(* CoDeSys 2.3 library: TcSystemCX80xx.lib *)
(* Libraries: STANDARD.LIB 5.6.98 12:03:02, TcBase.lib 14.5.09 12:14:08, TcSystem.lib 27.2.12 15:08:36, TcUtilities.lib 2.3.12 19:25:40 *)

(* Global variable list: Global_Variables *)
VAR_GLOBAL
	eGlobalSUpsState	: E_S_UPS_State; (* current ups state of S-UPS *)
END_VAR

(* Data type *)
TYPE E_CX8090_LED : (
	eLED_GREEN_OFF,
	eLED_GREEN_ON,
	eLED_GREEN_FLASHING_Quick,
	eLED_GREEN_FLASHING_200ms,
	eLED_GREEN_FLASHING_500ms,
	eLED_GREEN_FLASHING_Pulse,
	eLED_RED_OFF:=20,
	eLED_RED_ON,
	eLED_RED_FLASHING_Quick,
	eLED_RED_FLASHING_200ms,
	eLED_RED_FLASHING_500ms,
	eLED_RED_FLASHING_Pulse,
	eLED_GREEN_RED_OFF:=100,
	eLED_GREEN_RED_FLASHING_200ms,
	eLED_GREEN_RED_FLASHING_500ms
);
END_TYPE

(* Data type *)
TYPE E_S_UPS_Mode : (
	eSUPS_WrPersistData_Shutdown,			(* in case of powerfailure: writing of persistent data + shutdown*)
	eSUPS_WrPersistData_NoShutdown,			(* in case of powerfailure: writing of persistent data, no shutdown*)
	eSUPS_ImmediateShutdown,				(* in case of powerfailure: skips writing of data, immediate shutdown*)
	eSUPS_CheckPowerStatus					(* in case of powerfailure: reports powerfailure without action (no writing, no shutdown) *)
);
END_TYPE

(* Data type *)
TYPE E_S_UPS_State : (
	eSUPS_StateInit := -1,
	eSUPS_PowerOK,
	eSUPS_PowerFailure,
	eSUPS_WritePersistentData,
	eSUPS_QuickShutdown,
	eSUPS_WaitForRecover,
	eSUPS_WaitForPowerOFF
);


END_TYPE

(* POU F_CX8090_LED_ERR, ST *)
FUNCTION F_CX8090_LED_ERR : INT
VAR_INPUT
	eMode	: E_CX8090_LED;
END_VAR
{library private}
VAR
	iAdr		: POINTER TO DWORD;
	UINT32Value	: DWORD;
END_VAR
F_CX8090_LED_ERR	:= eMode;

CASE eMode OF
	eLED_GREEN_OFF: 
		UINT32Value	:=0;

	eLED_GREEN_ON:
		UINT32Value	:=1;

	eLED_GREEN_FLASHING_Quick: 
		UINT32Value	:=2;

	eLED_GREEN_FLASHING_200ms: 
		UINT32Value	:=3;

	eLED_GREEN_FLASHING_500ms: 
		UINT32Value	:=16#F3;

	eLED_GREEN_FLASHING_Pulse: 
		UINT32Value	:=16#13;

	eLED_RED_OFF: 
		UINT32Value	:=0;

	eLED_RED_ON: 
		UINT32Value	:=16#1_0000;

	eLED_RED_FLASHING_Quick: 
		UINT32Value	:=16#2_0000;

	eLED_RED_FLASHING_200ms: 
		UINT32Value	:=16#3_0000;

	eLED_RED_FLASHING_500ms: 
		UINT32Value	:=16#F3_0000;

	eLED_RED_FLASHING_Pulse: 
		UINT32Value	:=16#13_0000;

	eLED_GREEN_RED_OFF:
		UINT32Value	:=0;

	eLED_GREEN_RED_FLASHING_200ms:
		UINT32Value	:=16#3_0003;

	eLED_GREEN_RED_FLASHING_500ms:
		UINT32Value	:=16#F3_00F3;
ELSE
	UINT32Value		:=0;
	F_CX8090_LED_ERR:=-1;
END_CASE

iAdr	:= 16#AA010114;
iAdr^	:= UINT32Value;
END_FUNCTION

(* POU F_CX8090_LED_WD, ST *)
FUNCTION F_CX8090_LED_WD :INT
VAR_INPUT
	eMode	: E_CX8090_LED;
END_VAR
{library private}
VAR
	iAdr  		: POINTER TO DWORD;
	UINT32Value	: DWORD;
END_VAR
F_CX8090_LED_WD := eMode;

CASE eMode OF
	eLED_GREEN_OFF: 
		UINT32Value	:=0;

	eLED_GREEN_ON:
		UINT32Value	:=1;

	eLED_GREEN_FLASHING_Quick: 
		UINT32Value	:=2;

	eLED_GREEN_FLASHING_200ms: 
		UINT32Value	:=3;

	eLED_GREEN_FLASHING_500ms: 
		UINT32Value	:=16#F3;

	eLED_GREEN_FLASHING_Pulse: 
		UINT32Value	:=16#13;

	eLED_RED_OFF: 
		UINT32Value	:=0;

	eLED_RED_ON: 
		UINT32Value	:=16#1_0000;

	eLED_RED_FLASHING_Quick: 
		UINT32Value	:=16#2_0000;

	eLED_RED_FLASHING_200ms: 
		UINT32Value	:=16#3_0000;

	eLED_RED_FLASHING_500ms: 
		UINT32Value	:=16#F3_0000;

	eLED_RED_FLASHING_Pulse: 
		UINT32Value	:=16#13_0000;

	eLED_GREEN_RED_OFF:
		UINT32Value	:=0;

	eLED_GREEN_RED_FLASHING_200ms:
		UINT32Value	:=16#3_0003;

	eLED_GREEN_RED_FLASHING_500ms:
		UINT32Value	:=16#F3_00F3;
ELSE
	UINT32Value		:=0;
	F_CX8090_LED_WD :=-1;
END_CASE

iAdr	:= 16#AA010110;
iAdr^	:= UINT32Value;
END_FUNCTION

(* POU F_CX80xx_Address, ST *)
FUNCTION F_CX80xx_Address:INT	(* Read Address switch ;Error -1 wrong CX Typ*)
VAR_INPUT
	iCX_Typ	: INT;		(*Typ of CX8000, only the number, CX8031 Typ = 8031 ...*)
END_VAR
{library private}
VAR
	iAdr  			: POINTER TO DWORD;
	UINT64Value		: DWORD;
	UINT64Value_1	: DWORD;
	UINT64Value_2	: DWORD;
	byAddress		: BYTE;
	i				: SINT;
	M_1				: BOOL;
END_VAR
iAdr		:= 16#AA000310;
UINT64Value := iAdr^;

CASE iCX_Typ OF
	8031, 8051:
		UINT64Value_1	:= 16#F-(16#F AND ROR(UINT64Value,16));
		UINT64Value_2	:= 16#F-(16#F AND ROR(UINT64Value,20));
		F_CX80xx_Address:= DWORD_TO_INT((UINT64Value_1*10+UINT64Value_2));

	8010, 8090, 8091, 8093, 8095:
		UINT64Value_2	:=16#3FF-(16#3FF AND ROR(UINT64Value,16));
		UINT64Value_1	:=0;
		FOR i:=0 TO 9 DO
			M_1 := GETBIT32(UINT64Value_2,i);
			IF M_1 THEN
				UINT64Value_1 := SETBIT32(UINT64Value_1,9-i);
			END_IF
		END_FOR
		F_CX80xx_Address := DWORD_TO_INT(UINT64Value_1);
ELSE
	F_CX80xx_Address := -1;
END_CASE
END_FUNCTION

(* POU F_GetVersionTcSystemCX80xx, ST *)
FUNCTION F_GetVersionTcSystemCX80xx : UINT
VAR_INPUT
	nVersionElement		:	INT;
END_VAR
(*
	Possible nVersionElement parameter:
	1	:	major number
	2	:	minor number
	3	:	revision number
*)
VAR
END_VAR
(* Version history:
Date        | Version    | created under      		| Author   		| Remark 
--------------------------------------------------------------------------------------------------------------------------------------------------------------------- 
2011/12/06  | 1.0.0      | V2.11.0 (Build 2040)		| ICh		    | first version
2012/04/13  | 1.0.1      | V2.11.0 (Build 2218)		| RV	      	| add LED
2012/04/17  | 1.0.2      | V2.11.0 (Build 2219)		| ICH	      	| adding Pulse to LED enum, cleanup
*) 
CASE nVersionElement OF
1:	(* major number *)
	F_GetVersionTcSystemCX80xx := 1;
2:	(* minor number *)
	F_GetVersionTcSystemCX80xx := 0;
3:	(* revision number *)
	F_GetVersionTcSystemCX80xx := 2;
ELSE
	F_GetVersionTcSystemCX80xx := 16#FFFF;
END_CASE
END_FUNCTION

(* POU FB_NT_QuickShutdown, ST *)
FUNCTION_BLOCK FB_NT_QuickShutdown
VAR_INPUT
	NETID				:T_AmsNetId;
	START				:BOOL;
	TMOUT				:TIME := DEFAULT_ADS_TIMEOUT;
END_VAR
VAR_OUTPUT
	BUSY				:BOOL;
	ERR					:BOOL;
	ERRID				:UDINT;
END_VAR
{library private}
VAR
	ADSWRTCTL1			:ADSWRTCTL;
	RisingEdge			:R_TRIG;
	DELAY				:DWORD := 16#FFFFFFFF;
END_VAR
RisingEdge(CLK:=START);

IF RisingEdge.Q THEN
	ADSWRTCTL1(	NETID := NETID,
					PORT := AMSPORT_R3_SYSSERV,
					ADSSTATE := ADSSTATE_POWERFAILURE,
					DEVSTATE := 0,
					LEN := SIZEOF(DELAY),
					SRCADDR :=ADR(DELAY),
					Write := TRUE,
					TMOUT := TMOUT
				);
ELSE
	ADSWRTCTL1( Write:=FALSE);
END_IF


BUSY := ADSWRTCTL1.BUSY;
ERR := ADSWRTCTL1.ERR;
ERRID := ADSWRTCTL1.ERRID;
END_FUNCTION_BLOCK

(* POU FB_S_UPS_CX80xx, ST *)
FUNCTION_BLOCK FB_S_UPS_CX80xx
VAR_INPUT
	sNetID					: T_AmsNetId 		:= ''; 								(* '' = local netid *)
	iPLCPort				: UINT 				:= AMSPORT_R0_PLC_RTS1;				(* PLC Runtime System for writing persistent data *)
	tTimeout				: TIME 				:= DEFAULT_ADS_TIMEOUT;				(* ADS Timeout *)
	eUpsMode				: E_S_UPS_Mode		:= eSUPS_WrPersistData_Shutdown;	(* UPS mode (w/wo writing persistent data, w/wo shutdown) *)
	ePersistentMode			: E_PersistentMode	:= SPDM_2PASS;						(* mode for writing persistent data *)
	tRecoverTime			: TIME 				:= T#10s;							(* ON time to recover from short power failure in mode eSUPS_WrPersistData_NoShutdown/eSUPS_CheckPowerStatus  *)
END_VAR
VAR_OUTPUT
	bPowerFailDetect		: BOOL;													(* TRUE while powerfailure is detected *)
	eState					: E_S_UPS_State		:= eSUPS_PowerOK;					(* current ups state *)
END_VAR
{library private}
VAR
	fbWritePersistentData	: FB_WritePersistentData;
	fbNT_QuickShutdown 		: FB_NT_QuickShutdown;
	dwTemp					: DWORD;
	WaitForOffTimer			: TON;
	bFirstCycle				: BOOL := TRUE;
	bPowerOKInFirstCycle	: BOOL := FALSE;
	iAdr 					: POINTER TO DWORD := 16#B78A4000;
END_VAR
(* monitor power state *)
dwTemp := iAdr^;
bPowerFailDetect := NOT dwTemp.0;

(* load check *)
IF bFirstCycle THEN
	bFirstCycle 			:= FALSE;
	bPowerOKInFirstCycle 	:= NOT bPowerFailDetect;
END_IF

(* UPS State Machine *)
CASE eState OF
eSUPS_PowerOK:
	IF bPowerFailDetect THEN
		eState := eSUPS_PowerFailure; 		(* report powerfailure *)
		WaitForOffTimer(IN := FALSE, PT := tRecoverTime);
	END_IF


eSUPS_PowerFailure:
	IF bPowerOKInFirstCycle THEN
		(* allow saving/shutdown because S-UPS is fully loaded *)
		CASE eUpsMode OF
		eSUPS_WrPersistData_Shutdown,			(* in case of powerfailure: writing of persistent data + shutdown *)
		eSUPS_WrPersistData_NoShutdown:			(* in case of powerfailure: writing of persistent data, no shutdown *)
			(* start writing of persistent data *)
			fbWritePersistentData(
				NETID	:= sNetID,
				PORT	:= iPLCPort,
				START	:= TRUE,
				TMOUT	:= tTimeout,
				MODE	:= ePersistentMode
			);
			eState := eSUPS_WritePersistentData;


		eSUPS_CheckPowerStatus:					(* in case of powerfailure: reports powerfailure without action (no writing, no shutdown) *)
			(* check if power recovers *)
			eState := eSUPS_WaitForRecover;


		eSUPS_ImmediateShutdown:				(* in case of powerfailure: skips writing of data, immediate shutdown *)
			(* start quick shutdown *)
			fbNT_QuickShutdown(
				NETID := sNetID,
				START := TRUE,
				TMOUT := tTimeout
			);
			eState := eSUPS_QuickShutdown;

		END_CASE
	ELSE
		(* don't allow saving/shutdown because S-UPS was not fully loaded, just wait for OFF *)
		eState := eSUPS_WaitForPowerOFF;
	END_IF

eSUPS_WritePersistentData:
	(* writing of persistent data *)
	fbWritePersistentData(START	:= FALSE);

	IF eUpsMode = eSUPS_WrPersistData_NoShutdown THEN
		IF NOT fbWritePersistentData.BUSY THEN
			fbWritePersistentData(START	:= FALSE);

			(* wait for OFF *)
			eState := eSUPS_WaitForRecover;
			WaitForOffTimer(IN := FALSE, PT := tRecoverTime);
		END_IF
	ELSE
		IF NOT fbWritePersistentData.BUSY THEN
			fbWritePersistentData(START	:= FALSE);

			(* start quick shutdown *)
			fbNT_QuickShutdown(
				NETID := sNetID,
				START := TRUE,
				TMOUT := tTimeout
			);
			eState := eSUPS_QuickShutdown;
		END_IF
	END_IF


eSUPS_WaitForRecover:
	WaitForOffTimer(IN := (NOT bPowerFailDetect));
	IF WaitForOffTimer.Q THEN
		eState := eSUPS_PowerOK; 		(* report powerOK *)
	END_IF


eSUPS_QuickShutdown:
	(* quick shutdown *)
	fbNT_QuickShutdown(START := FALSE);
	IF NOT fbNT_QuickShutdown.BUSY THEN
		fbNT_QuickShutdown(START := FALSE);

		(* wait for OFF *)
		eState := eSUPS_WaitForPowerOFF;
	END_IF


eSUPS_WaitForPowerOFF:
	(* wait for OFF *)
	eState := eSUPS_WaitForPowerOFF;

END_CASE

eGlobalSUpsState := eState;
END_FUNCTION_BLOCK
